// Brief: Instrument Ready
FUNCTION_BLOCK PUBLIC FB_SlaveCtrlInstruReady EXTENDS FB_SlaveArmCtrlBase
VAR_INPUT
END_VAR
VAR_OUTPUT
END_VAR
VAR
END_VAR

METHOD PUBLIC init : BOOL
VAR_IN_OUT CONSTANT
	i_slaveArm	:FB_SlaveArm;
END_VAR
VAR_IN_OUT 
	r_slaveArmCtrlCmd :ST_SlaveArmCtrlCmds;
END_VAR


VAR
	j:INT;
	maxJntErr:LREAL;
	jntCtrlErr:Vec7d;
END_VAR
// DO NOT hold last command
//m_holdLastCmds := checkToHoldLastCmds(i_slaveArm);

//init
SUPER^.Init(i_slaveArm,r_slaveArmCtrlCmd);
END_METHOD

END_FUNCTION_BLOCK

(* stored: Version 1.1.0.1, ProductVersion 3.1.4024.11
   POU FB_SlaveCtrlInstruReady: Id {b4863c0c-c549-4967-ab29-6a1152ef3cd8}, SpecialFunc None
   Method init: Id {2537cbc9-bbc0-4d20-a9bf-3a888748c955} *)
